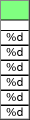
VISUALIZATION _VISU_WorkerDefGrid_VerifyHistory  // 30x120
VAR_IN_OUT
		m_Inst : FB_WorkerDefGrid_Verify;
END_VAR
    Rectangle (0,0 30x120)
    RoundedRectangle (0,0 30x20), colour toggle: m_Inst.bLastEject, invisible if: NOT m_Inst.tpShowResult.Q
    RoundedRectangle (0,30 30x15), "%d", tooltip "Ejected=1", text variable: m_Inst.nStateHistory[1], colour variable: m_Inst.nStateHistory_FillColor[1]
    RoundedRectangle (0,45 30x15), "%d", tooltip "Ejected=1", text variable: m_Inst.nStateHistory[2], colour variable: m_Inst.nStateHistory_FillColor[2]
    RoundedRectangle (0,60 30x15), "%d", tooltip "Ejected=1", text variable: m_Inst.nStateHistory[3], colour variable: m_Inst.nStateHistory_FillColor[3]
    RoundedRectangle (0,75 30x15), "%d", tooltip "Ejected=1", text variable: m_Inst.nStateHistory[4], colour variable: m_Inst.nStateHistory_FillColor[4]
    RoundedRectangle (0,90 30x15), "%d", tooltip "Ejected=1", text variable: m_Inst.nStateHistory[5], colour variable: m_Inst.nStateHistory_FillColor[5]
    RoundedRectangle (0,105 30x15), "%d", tooltip "Ejected=1", text variable: m_Inst.nStateHistory[6], colour variable: m_Inst.nStateHistory_FillColor[6]
END_VISUALIZATION

(* stored: Version 1.1.0.1, ProductVersion 3.1.4024.11
   Visu _VISU_WorkerDefGrid_VerifyHistory: Id {68e8549e-e731-41ad-b697-8276837995b9} *)
